{attribute 'linkalways'} 
{attribute 'no_explicit_call' := 'This FB is a CLASS and must be accessed using methods or properties'}
{attribute 'enable_dynamic_creation'}
FUNCTION_BLOCK _Array0to1OfLREAL EXTENDS ArrayDatatypeBase_1D
VAR CONSTANT
	lBound : DINT := 0;
	uBound : DINT := 1;
END_VAR
VAR
	localData : ARRAY [lBound..uBound] OF LREAL;
	activeData : REFERENCE TO ARRAY [lBound..uBound] OF LREAL REF= localData;
	elements : ARRAY [lBound..uBound] OF _LREAL(0.0);
	baseType : _LREAL(0.0);
END_VAR

PROPERTY PUBLIC Address : PVOID
GET
Address := ADR(activeData);
END_GET
END_PROPERTY

PROPERTY PUBLIC BaseDatatype : I_Datatype
GET
BaseDatatype := baseType;
END_GET
END_PROPERTY

METHOD PUBLIC ClearReference
VAR_INPUT
END_VAR
activeData REF= localData;
SetElementReference();
END_METHOD

METHOD PUBLIC Clone : I_Datatype
VAR
    pClone : POINTER TO _Array0to1OfLREAL;
END_VAR
pClone := __NEW(_Array0to1OfLREAL());
pClone^.Value := Value;
Clone := pClone^;
END_METHOD

METHOD FB_init : BOOL
VAR_INPUT
	bInitRetains : BOOL; // if TRUE, the retain variables are initialized (warm start / cold start)
	bInCopyCode : BOOL;  // if TRUE, the instance afterwards gets moved into the copy code (online change)
END_VAR
SetElementReference();
END_METHOD

METHOD PUBLIC MakeReferenceTo
VAR_INPUT
	ReferenceTarget : REFERENCE TO ARRAY [lBound..uBound] OF LREAL;
END_VAR
activeData REF= ReferenceTarget;
SetElementReference();
END_METHOD

METHOD PROTECTED OnSerializeArrayValues
VAR_INPUT
	Serializer : I_Serializer;
END_VAR
VAR
	i : DINT;
END_VAR
FOR i := lBound TO uBound DO
	elements[i].SerializeWith(Serializer);
END_FOR
END_METHOD

METHOD PROTECTED SetElementReference
VAR_INPUT
END_VAR
VAR
	i : DINT;
END_VAR
FOR i := lBound TO uBound DO
	elements[i].MakeReferenceTo(activeData[i]);
END_FOR
END_METHOD

PROPERTY PUBLIC Size : UDINT
GET
Size := SIZEOF(activeData);
END_GET
END_PROPERTY

METHOD PROTECTED TryDeserializeArrayValues : BOOL
VAR_INPUT
	Deserializer : I_Deserializer;
	Feedback : I_DeserializerFeedback;
END_VAR
VAR
	enumerator : I_DeserializerArrayForwardEnumerator;
	i : DINT;
END_VAR
enumerator := Deserializer.GetArrayEnumerator();
i := lBound;

WHILE enumerator.MoveNext() AND i <= uBound DO
	
	IF NOT elements[i].TryDeserializeFrom(enumerator.Current, Feedback) THEN
		EXIT;
	END_IF
	i := i + 1;

END_WHILE
enumerator.Dispose();
END_METHOD

METHOD PUBLIC TryGetElementAsDatatypeByIndex : BOOL
VAR_INPUT
	Index : DINT;
	Destination : REFERENCE TO I_Datatype;
END_VAR
IF Index < lbound OR Index > ubound THEN
	RETURN;
END_IF

Destination := elements[Index];
TryGetElementAsDatatypeByIndex := TRUE;
END_METHOD

METHOD PUBLIC TryGetLowerBound : BOOL
VAR_INPUT
	Dimention : UDINT;
	Destination : REFERENCE TO DINT;
END_VAR
IF Dimention = 1 THEN
	Destination := lBound;
	TryGetLowerBound := TRUE;
END_IF
END_METHOD

METHOD PUBLIC TryGetUpperBound : BOOL
VAR_INPUT
	Dimention : UDINT;
	Destination : REFERENCE TO DINT;
END_VAR
IF Dimention = 1 THEN
	Destination := uBound;
	TryGetUpperBound := TRUE;
END_IF
END_METHOD

METHOD TryMakeReferenceTo : BOOL
VAR_INPUT
	Target : I_Datatype;
END_VAR
VAR
	targetAsArray : I_ArrayDatatype;
	pTargetData : POINTER TO ARRAY [lBound..uBound] OF LREAL;
END_VAR
IF NOT Target.TryResolveAsArrayDatatype(targetAsArray) THEN
	RETURN;
END_IF

IF NOT (targetAsArray.Identifier = Identifier) THEN
	RETURN;
END_IF

pTargetData := Target.Address;
activeData REF= pTargetData^;
SetElementReference();
TryMakeReferenceTo := TRUE;
END_METHOD

PROPERTY PUBLIC Value : REFERENCE TO ARRAY [lBound..uBound] OF LREAL;
GET
Value ref= activeData;
END_GET
END_PROPERTY

END_FUNCTION_BLOCK

(* stored: Version 1.1.0.1, ProductVersion 3.1.4024.13
   POU _Array0to1OfLREAL: Id {918abd4d-9226-0a1c-0eea-38952724ed8c}, SpecialFunc None
   Folder Core: Id {cae6ca1d-fc09-0c26-2700-bb194bbfb108}
   Folder Constructor: Id {49a2ccde-3504-0b30-3d61-2889d0edc5d6}
   Folder Protected: Id {7aafcde4-93cf-0bcb-171c-c4e7817e2c7f}
   Folder Customize: Id {adcb4046-18b0-063f-3e9b-144224988397}
   Property Address: Id {de055903-e10b-0801-21f4-968458ef7053}
   Get Get: Id {23426e1b-911c-04ec-2c28-4f915e0616af}
   Property BaseDatatype: Id {f750c2a7-431e-067f-06d4-839fb9ab7d48}
   Get Get: Id {eebec1a9-21f9-047e-0fbc-05dfef4fdba0}
   Method ClearReference: Id {095bdce4-9009-092e-1851-9a9ab13a4035}
   Method Clone: Id {a67ebb1f-5873-0728-3872-9926894c0fb7}
   Method FB_init: Id {cd2bb5f4-1616-0348-0c6e-9237aa467d60}
   Method MakeReferenceTo: Id {6267e913-8559-00b9-35f7-fded6afaf6af}
   Method OnSerializeArrayValues: Id {557d2436-6d25-0c45-32f4-b7821ae54a48}
   Method SetElementReference: Id {96dedde8-ea5b-0254-31f3-21be16967f8a}
   Property Size: Id {39ca35df-0b93-01d2-3bba-c3cfb8016cf2}
   Get Get: Id {a8de7b97-d910-0643-1d46-031f1b533105}
   Method TryDeserializeArrayValues: Id {d2c4d5e6-7fbb-0698-1a3a-a9902c73dee4}
   Method TryGetElementAsDatatypeByIndex: Id {410c9b10-9462-0d20-0884-ffc2670ecb31}
   Method TryGetLowerBound: Id {542c9417-84c8-0f6c-3644-5c79864fbfa4}
   Method TryGetUpperBound: Id {6c84b8b7-d38f-0ba7-12a2-3d1942217367}
   Method TryMakeReferenceTo: Id {dd75f018-816c-068f-1642-7c5218b4ac66}
   Property Value: Id {f4c85a4e-8e8d-001f-02b8-9723623c642a}
   Get Get: Id {b6537905-a92c-0edf-0bfe-5264a5b98d4d} *)
